{attribute 'TcGenerated'}
{attribute 'no-analysis'}
{attribute 'linkalways'}
// This function has been automatically generated from the project information.
VAR_GLOBAL CONSTANT
	{attribute 'const_non_replaced'}
	stLibVersion_FsCommon : ST_LibVersion := (iMajor := 0, iMinor := 6, iBuild := 0, iRevision := 0, nFlags := 0, sVersion := '0.6.0');
END_VAR

(* stored: Version 1.1.0.1
   GVL Global_Version: Id {245431c4-a95b-05d4-388d-c273eeef5fc0} *)
